# EPICS autosave request: ADAndorIstar/andorIstarApp/Db/auto_settings.req
file "ADBase_settings.req",       P=$(P),  R=cam1:
file "andorIstar_settings.req",   P=$(P),  R=cam1:
file "NDFile_settings.req",       P=$(P),  R=cam1:
file "NDPluginBase_settings.req", P=$(P),  R=image1:
file "NDStdArrays_settings.req",  P=$(P),  R=image1:
#file "commonPlugin_settings.req", P=$(P)
# Comment out the following line on Linux or if there is no Shamrock spectrograph on Windows
#file "shamrock_settings.req",     P=$(P),  R=sham1:
